// TIA Portal V16 export
// export: Created 2021-09-08T12:46:14.8492597Z, ExportSetting WithDefaults, DisplayName Totally Integrated Automation Portal, DisplayVersion V16 Update 3, DisplayName TIA Portal Version Control Interface, DisplayVersion V16 Update 2, DisplayName TIA Portal Openness, DisplayVersion V16 Update 3, DisplayName TIA Portal Teamcenter Gateway, DisplayVersion V16, DisplayName STEP 7 Professional, DisplayVersion V16 Update 3, DisplayName STEP 7 Safety, DisplayVersion V16, DisplayName WinCC Advanced, DisplayVersion V16 Update 3
DATA_BLOCK "dtParmUF"   // DB26
{ S7_Optimized_Access := 'FALSE' }
VERSION : 0.1
// stored: AutoNumber true, DBAccessibleFromOPCUA true, IsOnlyStoredInLoadMemory false, IsWriteProtectedInAS false
   VAR RETAIN
      errSettingsLev : Bool;
      filtrationTime : UInt := 10;
      filtrateStartLevUF1 : Real;
      filtrateStopLevUF1 : Real;
      filtrateStartLevUF2 : Real;
      filtrateStopLevUF2 : Real;
      valHDP_ForHW : Real := 1.5;
      minFiltrLevForWash : Real := 50.0;
      delayHDP : UInt := 15;
      maxNumbHW_ByHDP : UInt := 3;
      HW_ToCEB1 : UInt := 3;
      HW_ToCEB2 : UInt := 6;
   END_VAR
BEGIN
END_DATA_BLOCK
